Fanuc KAREL source: kb00081.KL

-- PROVISIONAL review KL for V770-1; original PC SHA256 9c7c37b37536821580baa8e1ab5919656cef702a33e335aa6da874ed6c0f9877
-- Incomplete behavior may be omitted. Consult companion uncertainty JSON. Do not deploy.
PROGRAM KB00081
%NOLOCKGROUP
BEGIN
  -- UNRESOLVED_PC offsets 5-12; opcodes 9D,23
  -- UNRESOLVED_PC offsets 17-24; opcodes 9D,23
  -- UNRESOLVED_PC offsets 29-36; opcodes 9D,23
  -- UNRESOLVED_PC offsets 41-69; opcodes 27,22,22,22,31,23
  -- UNRESOLVED_PC offsets 74-78; opcodes 7F
END KB00081
